FUNCTION_BLOCK RemoteTriggeredLClock (* Used to initialize/update a time stamp remotely. The time stamp output is updated upon every REQ event *)
  (* Standard: 61499-2 *)
  (* Version 1.0, 2017-08-25, Marc Jakobi, HTW Berlin *)
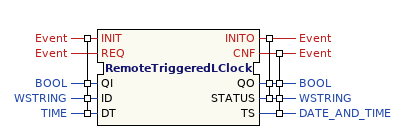
  EVENT_INPUT
    INIT WITH QI, ID, DT; (* Initialization Request *)
    REQ; (* Release Event *)
  END_EVENT
  EVENT_OUTPUT
    INITO WITH QO, STATUS; (* Initialization Confirm *)
    CNF WITH QO, TS, STATUS; (* Service Indication *)
  END_EVENT
  VAR_INPUT
    QI : BOOL; (* Input event qualifier *)
    ID : WSTRING; (* Connection identifier *)
    DT : TIME := T#1s; (* Internal clock's tick rate *)
  END_VAR
  VAR_OUTPUT
    QO : BOOL; (* Output event qualifier *)
    STATUS : WSTRING; (* Service status *)
    TS : DATE_AND_TIME; (* Time stamp *)
  END_VAR
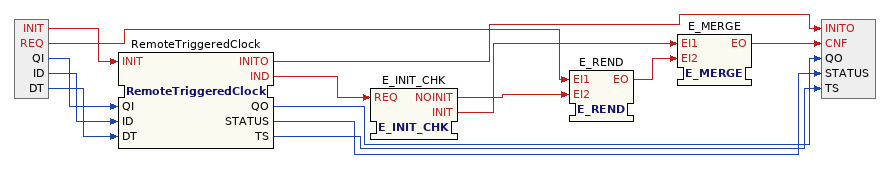
  FBS
    E_REND : E_REND;
    E_INIT_CHK : E_INIT_CHK;
    E_MERGE : E_MERGE;
    RemoteTriggeredClock : RemoteTriggeredClock;
  END_FBS
  EVENT_CONNECTIONS
    REQ TO E_REND.EI1;
    E_INIT_CHK.NOINIT TO E_REND.EI2;
    E_MERGE.EO TO CNF;
    E_INIT_CHK.INIT TO E_MERGE.EI1;
    E_REND.EO TO E_MERGE.EI2;
    INIT TO RemoteTriggeredClock.INIT;
    RemoteTriggeredClock.INITO TO INITO;
    RemoteTriggeredClock.IND TO E_INIT_CHK.REQ;
  END_CONNECTIONS
  DATA_CONNECTIONS
    QI TO RemoteTriggeredClock.QI;
    ID TO RemoteTriggeredClock.ID;
    DT TO RemoteTriggeredClock.DT;
    RemoteTriggeredClock.QO TO QO;
    RemoteTriggeredClock.TS TO TS;
    RemoteTriggeredClock.STATUS TO STATUS;
  END_CONNECTIONS
END_FUNCTION_BLOCK
